{attribute 'GeneratedUsingTerminal: AT2041-0250-0018'}
{attribute addProperty BoxType "AT2041-0250-0018"}
{attribute addProperty Id "A_0104_AT2042_5250_0019_AT2042_5250AT2042_33A3DF1B80"}
{attribute addProperty CRC "1399128306"}
{attribute addProperty Size "80"}
TYPE A_0040_AT2041_0250_0018_536500F2 EXTENDS AT2041_2EA6C9BF :
STRUCT
	{attribute addProperty Name "A_0104(AT2042-5250-0019) (AT2042-5250)"}
	{attribute addProperty PreviousPort "A_0040(AT2041-0250-0018) : B"}
	A_0104_AT2042_5250_0019_AT2042_5250 : AT2042_33A3DF1B;
END_STRUCT
END_TYPE

(* stored: Version 1.2.0.0, ProductVersion 3.1.4024.9
   DUT A_0040_AT2041_0250_0018_536500F2: Id {86634004-8e41-429e-a65c-233caf4b2e8e} *)
